PROGRAM AxisStop
VAR
	i				:USINT := 1;
END_VAR

// 所有轴停止
IF bAxis_All_Stop THEN
	FOR i:=1 TO nAxisNum DO
		aAxis_All_Stop_Group[i]^ := TRUE;
	END_FOR
ELSE
	FOR i:=1 TO nAxisNum DO
		aAxis_All_Stop_Group[i]^ := FALSE;
	END_FOR
END_IF

// LeftArm_Left_McStop
axis_LeftArm_Left_McStop(
	Axis:= axis_LeftArm_Left, 
	Execute:= bAxis_LeftArm_Left_McStop, 
	Deceleration:= , 
	Jerk:= , 
	Options:= , 
	Done=> , 
	Busy=> , 
	Active=> , 
	CommandAborted=> , 
	Error=> , 
	ErrorID=> );
	
// LeftArm_Right_McStop
axis_LeftArm_Right_McStop(
	Axis:= axis_LeftArm_Right, 
	Execute:= bAxis_LeftArm_Right_McStop, 
	Deceleration:= , 
	Jerk:= , 
	Options:= , 
	Done=> , 
	Busy=> , 
	Active=> , 
	CommandAborted=> , 
	Error=> , 
	ErrorID=> );
	
// LeftArm_Wrist_McStop	
axis_LeftArm_Wrist_McStop(
	Axis:= axis_LeftArm_Wrist, 
	Execute:= bAxis_LeftArm_Wrist_McStop, 
	Deceleration:= , 
	Jerk:= , 
	Options:= , 
	Done=> , 
	Busy=> , 
	Active=> , 
	CommandAborted=> , 
	Error=> , 
	ErrorID=> );

// LeftArm_Lift_McStop		
axis_LeftArm_Lift_McStop(
	Axis:= axis_LeftArm_Lift, 
	Execute:= bAxis_LeftArm_Lift_McStop, 
	Deceleration:= , 
	Jerk:= , 
	Options:= , 
	Done=> , 
	Busy=> , 
	Active=> , 
	CommandAborted=> , 
	Error=> , 
	ErrorID=> );

	
// RightArm_Left_McStop
axis_RightArm_Left_McStop(
	Axis:= axis_RightArm_Left, 
	Execute:= bAxis_RightArm_Left_McStop, 
	Deceleration:= , 
	Jerk:= , 
	Options:= , 
	Done=> , 
	Busy=> , 
	Active=> , 
	CommandAborted=> , 
	Error=> , 
	ErrorID=> );
	
// RightArm_Right_McStop
axis_RightArm_Right_McStop(
	Axis:= axis_RightArm_Right, 
	Execute:= bAxis_RightArm_Right_McStop, 
	Deceleration:= , 
	Jerk:= , 
	Options:= , 
	Done=> , 
	Busy=> , 
	Active=> , 
	CommandAborted=> , 
	Error=> , 
	ErrorID=> );
	
// RightArm_Wrist_McStop	
axis_RightArm_Wrist_McStop(
	Axis:= axis_RightArm_Wrist, 
	Execute:= bAxis_RightArm_Wrist_McStop, 
	Deceleration:= , 
	Jerk:= , 
	Options:= , 
	Done=> , 
	Busy=> , 
	Active=> , 
	CommandAborted=> , 
	Error=> , 
	ErrorID=> );

// RightArm_Lift_McStop		
axis_RightArm_Lift_McStop(
	Axis:= axis_RightArm_Lift, 
	Execute:= bAxis_RightArm_Lift_McStop, 
	Deceleration:= , 
	Jerk:= , 
	Options:= , 
	Done=> , 
	Busy=> , 
	Active=> , 
	CommandAborted=> , 
	Error=> , 
	ErrorID=> );

// BigGate_Left_McStop	
axis_BigGate_Left_McStop(
	Axis:= axis_BigGate_Left, 
	Execute:= bAxis_BigGate_Left_McStop, 
	Deceleration:= , 
	Jerk:= , 
	Options:= , 
	Done=> , 
	Busy=> , 
	Active=> , 
	CommandAborted=> , 
	Error=> , 
	ErrorID=> );
	
// BigGate_Right_McStop
axis_BigGate_Right_McStop(
	Axis:= axis_BigGate_Right, 
	Execute:= bAxis_BigGate_Right_McStop, 
	Deceleration:= , 
	Jerk:= , 
	Options:= , 
	Done=> , 
	Busy=> , 
	Active=> , 
	CommandAborted=> , 
	Error=> , 
	ErrorID=> );
	
// SmallGate_Left_McStop	
axis_SmallGate_Left_McStop(
	Axis:= axis_SmallGate_Left, 
	Execute:= bAxis_SmallGate_Left_McStop, 
	Deceleration:= , 
	Jerk:= , 
	Options:= , 
	Done=> , 
	Busy=> , 
	Active=> , 
	CommandAborted=> , 
	Error=> , 
	ErrorID=> );
	
// SmallGate_Right_McStop
axis_SmallGate_Right_McStop(
	Axis:= axis_SmallGate_Right, 
	Execute:= bAxis_SmallGate_Right_McStop, 
	Deceleration:= , 
	Jerk:= , 
	Options:= , 
	Done=> , 
	Busy=> , 
	Active=> , 
	CommandAborted=> , 
	Error=> , 
	ErrorID=> );
	
	
// BackGate_Left_McStop	
axis_BackGate_Left_McStop(
	Axis:= axis_BackGate_Left, 
	Execute:= bAxis_BackGate_Left_McStop, 
	Deceleration:= , 
	Jerk:= , 
	Options:= , 
	Done=> , 
	Busy=> , 
	Active=> , 
	CommandAborted=> , 
	Error=> , 
	ErrorID=> );
	
// BackGate_Right_McStop
axis_BackGate_Right_McStop(
	Axis:= axis_BackGate_Right, 
	Execute:= bAxis_BackGate_Right_McStop, 
	Deceleration:= , 
	Jerk:= , 
	Options:= , 
	Done=> , 
	Busy=> , 
	Active=> , 
	CommandAborted=> , 
	Error=> , 
	ErrorID=> );

END_PROGRAM

(* stored: Version 1.1.0.1, ProductVersion 3.1.4024.14
   POU AxisStop: Id {d8bac268-a103-4f37-a01b-e341c61b0e22}, SpecialFunc None *)
